TYPE ST_HMI_MapItem : 
STRUCT
	sName: WSTRING(127);
	sDescription: WSTRING(127);
	sPosition: WSTRING(127);
	nStatus: INT;
END_STRUCT
END_TYPE

(* stored: DUT ST_HMI_MapItem: Id 3adf780c-5d7f-4102-ac4d-676e9aa7558a *)
